FUNCTION_BLOCK SoEResetTestSuite
VAR
	StubAxis : AXIS_REF;
	iStubTask : I_Task;
	Soe_Reset : SoEResetTask;
	TestObjRunner : ObjectRunner<99>;
	ObjTestSuite : TestSuite<TestSuiteParameter.MaxTestCount>(ResultFile := JUnitResultFile) := (TestSuiteName := 'Object Test Suite');
END_VAR

TaskRejectsCycleCallWithoutAxisRef_Test();
TaskAcceptsResetCommand_Test();
TaskRejectsDuplicateResetCommand_Test();
CheckCorrectRegistration_Test();

METHOD CheckCorrectRegistration_Test : BOOL
VAR_INST
	Expected : BOOL := TRUE;
	Actual	 : BOOL;
END_VAR
IF ObjTestSuite.Test(__POUNAME()).ExecuteTest() THEN
	Soe_Reset.RegisterWithParent(TestObjRunner);
	Actual := TestObjRunner.CyclicModuleCount = TestObjRunner.AbortableModuleCount AND
				TestObjRunner.CyclicModuleCount = TestObjRunner.TaskModuleCount AND
				TestObjRunner.CyclicModuleCount = TestObjRunner.ResettableModuleCount;
	ObjTestSuite.Test(__POUNAME()).AssertEqual(Expected, Actual);
END_IF
END_METHOD

METHOD TaskAcceptsResetCommand_Test : BOOL
VAR_INST
	Expected : BOOL := TRUE;
	Actual	 : BOOL;
END_VAR
IF ObjTestSuite.Test(__POUNAME()).ExecuteTest() THEN
	Actual := SUCCEEDED(Soe_Reset.Reset());
	Soe_Reset.Abort();
	ObjTestSuite.Test(__POUNAME()).AssertEqual(Expected, Actual);
END_IF
END_METHOD

METHOD TaskRejectsCycleCallWithoutAxisRef_Test
VAR_INST
	Expected : BOOL := TRUE;
	Actual	 : BOOL;
END_VAR
IF ObjTestSuite.Test(__POUNAME()).ExecuteTest() THEN
	Actual := FAILED(Soe_Reset.Cycle());
	Soe_Reset.AxisRef REF= StubAxis;
	ObjTestSuite.Test(__POUNAME()).AssertEqual(Expected, Actual);
END_IF
END_METHOD

METHOD TaskRejectsDuplicateResetCommand_Test : BOOL
VAR_INST
	Expected : BOOL := TRUE;
	Actual	 : BOOL;
END_VAR
IF ObjTestSuite.Test(__POUNAME()).ExecuteTest() THEN
	Soe_Reset.Reset();
	Actual := FAILED(Soe_Reset.Reset());
	Soe_Reset.Abort();
	ObjTestSuite.Test(__POUNAME()).AssertEqual(Expected, Actual);
END_IF
END_METHOD

END_FUNCTION_BLOCK

(* stored: Version 1.1.0.1
   POU SoEResetTestSuite: Id {51229c30-760a-4dc9-943c-9ac0c10638e5}, SpecialFunc None
   Method CheckCorrectRegistration_Test: Id {6e5c4cac-4975-4991-8748-3fa4bd23314a}
   Method TaskAcceptsResetCommand_Test: Id {e9903409-a92e-4aaf-996b-b34d77337a77}
   Method TaskRejectsCycleCallWithoutAxisRef_Test: Id {7e5f0857-ff2e-4d82-9bac-48352d060a7f}
   Method TaskRejectsDuplicateResetCommand_Test: Id {929b7d0a-5392-4603-aaa4-4d618865beeb} *)
